// TwinCAT 3 PLC project SPS
// ProgramVersion: 3.1.4026.10
// libraries:
//   Tc2_Standard, * (Beckhoff Automation GmbH)
//   Tc2_System, * (Beckhoff Automation GmbH)
//   Tc3_Vision, * (Beckhoff Automation GmbH)
// project tree:
//   / PlcTask.TcTTO
//   POUs/ Ablage.TcPOU, Beispiel_FindContours.TcPOU, MAIN.TcPOU

CONFIGURATION SPS
    RESOURCE PLC ON TwinCAT3
        TASK PlcTask(INTERVAL := T#10ms, PRIORITY := 20);
        PROGRAM MAIN WITH PlcTask : MAIN;
    END_RESOURCE
END_CONFIGURATION

// ---- POUs/MAIN.TcPOU
PROGRAM MAIN
VAR
	fbCamera_2					:FB_VN_SimpleCameraControl;
	eState_2					:ETcVnCameraState; 
	
	hr                    :    HRESULT; 
	
	ipImageIn             :    ITcVnImage;
	ipImageInDisp         :    ITcVnDisplayableImage;
	ipImageWork           :    ITcVnImage;
	ipImageThresholdDisp  :    ITcVnDisplayableImage;
	ipImageRes            :    ITcVnImage;
	ipImageResDisp        :    ITcVnDisplayableImage;
	
	// Sample Specific Variables    
	ipContourList         :    ITcVnContainer;
	ipContourResultList   :    ITcVnContainer;
	ipContour             :    ITcVnContainer;
	ipIterator            :    ITcVnForwardIterator;
	aOffset               :    TcVnPoint;
	
	fThreshold            :    LREAL := 70;
	
	fArea                 :    LREAL;
	fAreaMin              :    LREAL := 100;
	fAreaMax              :    LREAL := 100000;
	
	fCircularity          :    LREAL;
	fCircularityMin       :    LREAL := 0.8;
	
	// Image Infos
	stPixelFormat         :    TcVnPixelFormat;
	
	// COLORS
	aColorGreen           :    TcVnVector4_LREAL    :=    [0, 255, 0];
END_VAR

eState_2 := fbCamera_2.GetState();

IF eState_2 = TCVN_CS_ERROR THEN
	hr := fbCamera_2.Reset();
	
ELSIF eState_2 < TCVN_CS_ACQUIRING THEN
	hr := fbCamera_2.StartAcquisition();
	
ELSIF eState_2 = TCVN_CS_ACQUIRING THEN
	hr := fbCamera_2.GetCurrentImage(ipImageIn);
	
	IF SUCCEEDED(hr) AND ipImageIn <> 0 THEN
		// Image Segementation
		hr := F_VN_Threshold(ipImageIn, ipImageWork, fThreshold, 255, TCVN_TT_Binary, hr);
		
		// Find Contours
		hr := F_VN_FindContoursExp(
				ipSrcImage             := ipImageWork, 
				ipContours             := ipContourList, 
				eRetrievalMode         := ETcVnContourRetrievalmode.TCVN_CRM_LIST, 
				eApproximationMethod   := ETcVnContourApproximationMethod.TCVN_CAM_SIMPLE, 
				aOffset                := aOffset, 
				hrPrev                 := hr);
				
		// Filter Contours
		hr := F_VN_GetForwardIterator(ipContourList, ipIterator, hr);
		hr := F_VN_CreateContainer(ipContourResultList, ContainerType_Vector_Vector_TcVnPoint2_DINT, 0, hr);
		
		WHILE SUCCEEDED(hr) AND_THEN ipIterator.CheckIfEnd() <> S_OK DO
		
			hr := F_VN_GetContainer(ipIterator, ipContour, hr);
			hr := F_VN_IncrementIterator(ipIterator, hr);
		
			// Filter by Area
			hr := F_VN_ContourArea(ipContour, fArea, hr);
		
			IF fArea > fAreaMin AND fArea < fAreaMax THEN
		
				// Filter by Circularity
				hr := F_VN_ContourCircularity(ipContour, fCircularity, hr);
		
				IF fCircularity > fCircularityMin THEN
					// Add contour to the result contour container
					hr := F_VN_AppendToContainer_ITcVnContainer(ipContour, ipContourResultList, hr);
		
				END_IF
			END_IF
		END_WHILE
		
		// Draw contours into the result image and display it
		hr := F_VN_DrawContours(ipContourResultList, -1, ipImageRes, aColorGreen, 3, hr);
		hr := F_VN_TransformIntoDisplayableImage(ipImageRes, ipImageResDisp, hr);
	END_IF
END_IF

END_PROGRAM

// ---- POUs/Ablage.TcPOU
PROGRAM Ablage
VAR
	hr							:HRESULT;
	fbCamera					:FB_VN_SimpleCameraControl;
	eState						:ETcVnCameraState; 
	ipImageIn					:ITcVnImage;
	ipFilteredImage				:ITcVnImage; 
	ipProcessedImage			:ITcVnImage; 
	ipImageInDisplay			:ITcVnDisplayableImage; 
	ipFilteredImageToDisplay	:ITcVnDisplayableImage; 
	ipProcessedImageToDisplay	:ITcVnDisplayableImage; 
	
	ipContainer  : ITcVnContainer;
	
	fThreshold					:LREAL := 140;
	
	aCenter    : TcVnPoint2_REAL;
    fRadius    : REAL := 30;
END_VAR

Beispiel_FindContours();

eState := fbCamera.GetState();

IF eState = TCVN_CS_ERROR THEN
	hr := fbCamera.Reset();
	
ELSIF eState < TCVN_CS_ACQUIRING THEN
	hr := fbCamera.StartAcquisition();
	
ELSIF eState = TCVN_CS_ACQUIRING THEN
	hr := fbCamera.GetCurrentImage(ipImageIn);
	
	IF SUCCEEDED(hr) AND ipImageIn <> 0 THEN
		
		hr := F_VN_GaussianFilter(
			ipSrcImage 		:= ipImageIn,
			ipDestImage 	:= ipFilteredImage,
			nFilterWidth 	:= 3,
			nFilterHeight 	:= 3,
			hrPrev := hr);
		
		hr := F_VN_Threshold(
			ipSrcImage 		:= ipFilteredImage,	
			ipDestImage 	:= ipProcessedImage,
			fThreshold 		:= fThreshold,
			fMaxValue		:= 255,
			eThresholdType 	:= TCVN_TT_Binary,
			hrPrev 			:= hr);
			
		hr := F_VN_CreateContainer(ipContainer, ContainerType_Vector_ITcVnImage, 1, hr);
			
		hr := F_VN_AppendToContainer_ITcVnImage(
			ipElement 		:= ipProcessedImage,
			ipContainer 	:= ipContainer,
			hrPrev 			:= hr);
			
		hr := F_VN_EnclosingCircle(
				ipPointSet 	:= ipContainer,
				aCenter 	:= aCenter,
				fRadius 	:= fRadius,
				hrPrev 		:= hr);
				
			
		
		//hr := F_VN_TransformIntoDisplayableImage(ipImageIn, ipImageInDisplay, hr);
		//hr := F_VN_TransformIntoDisplayableImage(ipFilteredImage, ipFilteredImageToDisplay, hr);
		//hr := F_VN_TransformIntoDisplayableImage(ipProcessedImage, ipProcessedImageToDisplay, hr);
		
		
	END_IF

END_IF

END_PROGRAM

// ---- POUs/Beispiel_FindContours.TcPOU
PROGRAM Beispiel_FindContours
VAR
fbCamera_2					:FB_VN_SimpleCameraControl;
eState_2					:ETcVnCameraState; 

hr                    :    HRESULT; 

ipImageIn             :    ITcVnImage;
ipImageInDisp         :    ITcVnDisplayableImage;
ipImageWork           :    ITcVnImage;
ipImageThresholdDisp  :    ITcVnDisplayableImage;
ipImageRes            :    ITcVnImage;
ipImageResDisp        :    ITcVnDisplayableImage;

// Sample Specific Variables    
ipContourList         :    ITcVnContainer;
ipContourResultList   :    ITcVnContainer;
ipContour             :    ITcVnContainer;
ipIterator            :    ITcVnForwardIterator;
aOffset               :    TcVnPoint;

fThreshold            :    LREAL := 70;

fArea                 :    LREAL;
fAreaMin              :    LREAL := 100;
fAreaMax              :    LREAL := 100000;

fCircularity          :    LREAL;
fCircularityMin       :    LREAL := 0.8;

// Image Infos
stPixelFormat         :    TcVnPixelFormat;

// COLORS
aColorGreen           :    TcVnVector4_LREAL    :=    [0, 255, 0];
END_VAR

eState_2 := fbCamera_2.GetState();

IF eState_2 = TCVN_CS_ERROR THEN
	hr := fbCamera_2.Reset();
	
ELSIF eState_2 < TCVN_CS_ACQUIRING THEN
	hr := fbCamera_2.StartAcquisition();
	
ELSIF eState_2 = TCVN_CS_ACQUIRING THEN
	hr := fbCamera_2.GetCurrentImage(ipImageIn);
	
	IF SUCCEEDED(hr) AND ipImageIn <> 0 THEN
		// Image Segementation
		hr := F_VN_Threshold(ipImageIn, ipImageWork, fThreshold, 255, TCVN_TT_Binary, hr);
		
		// Find Contours
		hr := F_VN_FindContoursExp(
				ipSrcImage             := ipImageWork, 
				ipContours             := ipContourList, 
				eRetrievalMode         := ETcVnContourRetrievalmode.TCVN_CRM_LIST, 
				eApproximationMethod   := ETcVnContourApproximationMethod.TCVN_CAM_SIMPLE, 
				aOffset                := aOffset, 
				hrPrev                 := hr);
				
		// Filter Contours
		hr := F_VN_GetForwardIterator(ipContourList, ipIterator, hr);
		hr := F_VN_CreateContainer(ipContourResultList, ContainerType_Vector_Vector_TcVnPoint2_DINT, 0, hr);
		
		WHILE SUCCEEDED(hr) AND_THEN ipIterator.CheckIfEnd() <> S_OK DO
		
			hr := F_VN_GetContainer(ipIterator, ipContour, hr);
			hr := F_VN_IncrementIterator(ipIterator, hr);
		
			// Filter by Area
			hr := F_VN_ContourArea(ipContour, fArea, hr);
		
			IF fArea > fAreaMin AND fArea < fAreaMax THEN
		
				// Filter by Circularity
				hr := F_VN_ContourCircularity(ipContour, fCircularity, hr);
		
				IF fCircularity > fCircularityMin THEN
					// Add contour to the result contour container
					hr := F_VN_AppendToContainer_ITcVnContainer(ipContour, ipContourResultList, hr);
		
				END_IF
			END_IF
		END_WHILE
		
		// Draw contours into the result image and display it
		hr := F_VN_DrawContours(ipContourResultList, -1, ipImageRes, aColorGreen, 3, hr);
		hr := F_VN_TransformIntoDisplayableImage(ipImageRes, ipImageResDisp, hr);
	END_IF
END_IF

END_PROGRAM
